PROGRAM Initialize
VAR
	Initialize_RTrig: R_TRIG;
	iStep : INT;
END_VAR

Initialize_RTrig(CLK:= G_MachineControl.bInitialize);
IF Initialize_RTrig.Q THEN
	G_MachineControl.bInitializeDone := FALSE;
	iStep := 10;
END_IF

CASE iStep OF
	10:
		//G_Home.H10_bHome := TRUE;
		G_Home.H20_bHome := TRUE;
		iStep := 20;
		
	20:
		IF G_Home.H20_bHomeDone THEN
			G_MachineControl.bInitialize := FALSE;
			G_MachineControl.bInitializeDone := TRUE;
			iStep := 0;
		END_IF
END_CASE

//Hello World

END_PROGRAM

(* stored: Version 1.1.0.1, ProductVersion 3.1.4024.12
   POU Initialize: Id {f890748c-baff-401a-b907-3c39079f0807}, SpecialFunc None *)
